Omron CX-Programmer project NewProject (CX-Programmer 9.51)

# PLC my_first_project: CP1L L
; My first Project

## Global symbols (name address type ; comment)
W0.02 BOOL  ; comment

## Program NewProgram1 (cyclic task 0)
Local symbols
button_1 0.00 BOOL  ; comment
button_2 0.01 BOOL  ; comment
button_3 0.02 BOOL  ; comment
button_4 0.03 BOOL  ; comment
out_1 100.00 BOOL  ; out_1
out_2 100.01 BOOL  ; comment

### Section Section1

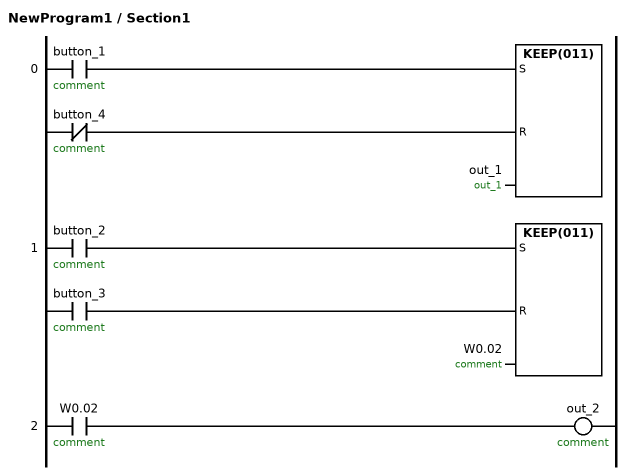
; rung 0
LD button_1  ; comment
LDNOT button_4  ; comment
KEEP(011) out_1  ; out_1
; rung 1
LD button_2  ; comment
LD button_3  ; comment
KEEP(011) W0.02  ; comment
; rung 2
LD W0.02  ; comment
OUT out_2  ; comment

### Section END
; rung 0
END(001)